FUNCTION_BLOCK FB_CylinderTemp EXTENDS FB_CylinderBase
VAR_INPUT
	fTempCurrent		AT %I*		:		LREAL;		// Hardware input signal: cylinder temperature
END_VAR
VAR_OUTPUT
END_VAR
VAR
END_VAR

END_FUNCTION_BLOCK

(* stored: Version 1.1.0.1, ProductVersion 3.1.4024.15
   POU FB_CylinderTemp: Id {853695ea-0a11-40ec-9858-19484fa1f60c}, SpecialFunc None *)
